(* CoDeSys 2.3.9.47 project: gym.prx *)
(* Libraries: TcBaseBX.lbx 10.5.06 08:50:20, TcSystemBX.lbx 11.6.12 13:56:16, standard.lbx 5.12.03 08:02:30, TcEIB.lbx 16.5.14 14:12:22, TcBABasicBX.lbx 22.7.15 15:46:56 *)

(* Task configuration *)
TASK Standard (PRIORITY := 0, INTERVAL := T#20ms);
	MAIN
END_TASK

(* Global variable list: KNX *)
VAR_GLOBAL
	fb_KL6301_0:								KL6301;


	fb_gym01_send_status_ex: 					EIB_BIT_SEND_EX;
	fb_gym02_send_status_ex: 					EIB_BIT_SEND_EX;
	fb_training01_send_status_ex: 				EIB_BIT_SEND_EX;
	fb_training02_send_status_ex: 				EIB_BIT_SEND_EX;
	fb_training03_send_status_ex: 				EIB_BIT_SEND_EX;
	fb_gym_stairs_bra_send_status_ex: 			EIB_BIT_SEND_EX;
	fb_pool_hall_spotlight_send_status_ex: 		EIB_BIT_SEND_EX;
	fb_pool_hall_LED_send_status_ex: 			EIB_BIT_SEND_EX;

	fb_pool_light_send_status_ex: 				EIB_BIT_SEND_EX;
	fb_sphere_ceiling_light_send_status_ex: 		EIB_BIT_SEND_EX;
	fb_sphere_light_send_status_ex: 			EIB_BIT_SEND_EX;
	fb_gym_cinema_bra_send_status_ex: 		EIB_BIT_SEND_EX;
	fb_gym_shower01_light_send_status_ex: 		EIB_BIT_SEND_EX;
	fb_gym_shower02_light_send_status_ex: 		EIB_BIT_SEND_EX;
	fb_gym_WC_corridor_send_status_ex: 		EIB_BIT_SEND_EX;
	fb_gym_stairs_light_send_status_ex: 			EIB_BIT_SEND_EX;

	fb_gym_WC_light_send_status_ex: 			EIB_BIT_SEND_EX;
	fb_training_light_send_status_ex: 			EIB_BIT_SEND_EX;
	fb_gym_light_send_status_ex: 				EIB_BIT_SEND_EX;

	fb_gym_all_send_status_ex: 				EIB_BIT_SEND_EX;
	fb_training_all_send_status_ex: 				EIB_BIT_SEND_EX;
	fb_training_1column_send_status_ex: 		EIB_BIT_SEND_EX;
	fb_pool_inwater_send_status_ex: 			EIB_BIT_SEND_EX;


	fb_outside_bigBulbs_send_status_ex:		EIB_BIT_SEND_EX;
	fb_outside_smallBulbs_send_status_ex:		EIB_BIT_SEND_EX;
	fb_outside_pingPongTable_send_status_ex:	EIB_BIT_SEND_EX;
	fb_outside_plantsLightning_send_status_ex:	EIB_BIT_SEND_EX;

	fb_pool_floor_heating_pump_send_status_ex:	EIB_BIT_SEND_EX;
	fb_gym_floor_heating_pump_send_status_ex:	EIB_BIT_SEND_EX;
	fb_vent_heating_pump_send_status_ex:		EIB_BIT_SEND_EX;
	fb_heating_pump_send_status_ex:			EIB_BIT_SEND_EX;


	fb_pool_floor_heating_pump_read:			EIB_BIT_REC ;
	fb_gym_floor_heating_pump_read:			EIB_BIT_REC ;
	fb_vent_heating_pump_read:				EIB_BIT_REC ;
	fb_heating_pump_read:					EIB_BIT_REC ;

	fb_gym01_read: 					EIB_BIT_REC;
	fb_gym02_read: 					EIB_BIT_REC;
	fb_training01_read:				EIB_BIT_REC;
	fb_training02_read:				EIB_BIT_REC;
	fb_training03_read:				EIB_BIT_REC;
	fb_gym_stairs_bra_read:			EIB_BIT_REC;
	fb_pool_hall_spotlight_read:		EIB_BIT_REC;
	fb_pool_hall_LED_read:			EIB_BIT_REC;

	fb_pool_light_read:				EIB_BIT_REC;
	fb_sphere_ceiling_light_read:		EIB_BIT_REC;
	fb_sphere_light_read:				EIB_BIT_REC;
	fb_gym_cinema_bra_read:			EIB_BIT_REC;
	fb_gym_shower01_light_read:		EIB_BIT_REC;
	fb_gym_shower02_light_read:		EIB_BIT_REC;
	fb_gym_WC_corridor_read:			EIB_BIT_REC;
	fb_gym_stairs_light_read:			EIB_BIT_REC;

	fb_gym_WC_light_read:			EIB_BIT_REC;
	fb_training_light_read:				EIB_BIT_REC;
	fb_gym_light_read:				EIB_BIT_REC;
	fb_outside_bigBulbs_read:			EIB_BIT_REC;
	fb_outside_smallBulbs_read:		EIB_BIT_REC;
	fb_outside_pingPongTable_read:	EIB_BIT_REC;
	fb_outside_plantsLightning_read:	EIB_BIT_REC;

	fb_gym_all_read: 					EIB_BIT_REC;
	fb_training_all_read: 				EIB_BIT_REC;
	fb_training_1column_read: 			EIB_BIT_REC;
	fb_pool_inwater_read: 				EIB_BIT_REC;

	gym_lights					:	BOOL;


(*2/0/x*)
	pool_floor_heating_pump_adr:								EIB_GROUP_ADDR :=(MAIN:=2, SUB_MAIN:=0, NUMBER:=1);
	gym_floor_heating_pump_adr:								EIB_GROUP_ADDR :=(MAIN:=2, SUB_MAIN:=0, NUMBER:=2);
	vent_heating_pump_adr:									EIB_GROUP_ADDR :=(MAIN:=2, SUB_MAIN:=0, NUMBER:=3);
	heating_pump_adr:										EIB_GROUP_ADDR :=(MAIN:=2, SUB_MAIN:=0, NUMBER:=4);

	pool_floor_heating_pump_status_adr:						EIB_GROUP_ADDR :=(MAIN:=2, SUB_MAIN:=0, NUMBER:=101);
	gym_floor_heating_pump_status_adr:							EIB_GROUP_ADDR :=(MAIN:=2, SUB_MAIN:=0, NUMBER:=102);
	vent_heating_pump_status_adr:								EIB_GROUP_ADDR :=(MAIN:=2, SUB_MAIN:=0, NUMBER:=103);
	heating_pump_staus_adr:									EIB_GROUP_ADDR :=(MAIN:=2, SUB_MAIN:=0, NUMBER:=104);


(*2/1/x*)
	gym01_adr:												EIB_GROUP_ADDR :=(MAIN:=2, SUB_MAIN:=1, NUMBER:=1);
	gym02_adr:												EIB_GROUP_ADDR :=(MAIN:=2, SUB_MAIN:=1, NUMBER:=2);
	training01_adr:											EIB_GROUP_ADDR :=(MAIN:=2, SUB_MAIN:=1, NUMBER:=3);
	training02_adr:											EIB_GROUP_ADDR :=(MAIN:=2, SUB_MAIN:=1, NUMBER:=4);
	training03_adr:											EIB_GROUP_ADDR :=(MAIN:=2, SUB_MAIN:=1, NUMBER:=5);
	gym_stairs_bra_adr:										EIB_GROUP_ADDR :=(MAIN:=2, SUB_MAIN:=1, NUMBER:=6);
	pool_hall_spotlight_adr:									EIB_GROUP_ADDR :=(MAIN:=2, SUB_MAIN:=1, NUMBER:=7);
	pool_hall_LED_adr:										EIB_GROUP_ADDR :=(MAIN:=2, SUB_MAIN:=1, NUMBER:=8);
	pool_light_adr:											EIB_GROUP_ADDR :=(MAIN:=2, SUB_MAIN:=1, NUMBER:=9);
	sphere_ceiling_light_adr:									EIB_GROUP_ADDR :=(MAIN:=2, SUB_MAIN:=1, NUMBER:=10);
	sphere_light_adr:											EIB_GROUP_ADDR :=(MAIN:=2, SUB_MAIN:=1, NUMBER:=11);
	gym_cinema_bra_adr:										EIB_GROUP_ADDR :=(MAIN:=2, SUB_MAIN:=1, NUMBER:=12);
	gym_shower01_light_adr:									EIB_GROUP_ADDR :=(MAIN:=2, SUB_MAIN:=1, NUMBER:=13);
	gym_shower02_light_adr:									EIB_GROUP_ADDR :=(MAIN:=2, SUB_MAIN:=1, NUMBER:=14);
	gym_WC_corridor_adr:										EIB_GROUP_ADDR :=(MAIN:=2, SUB_MAIN:=1, NUMBER:=15);
	gym_stairs_light_adr:										EIB_GROUP_ADDR:= (MAIN:=2, SUB_MAIN:=1, NUMBER:=16);
	gym_WC_light_adr:										EIB_GROUP_ADDR:= (MAIN:=2, SUB_MAIN:=1, NUMBER:=17);
	training_light_adr:											EIB_GROUP_ADDR:= (MAIN:=2, SUB_MAIN:=1, NUMBER:=18);
	gym_light_adr:											EIB_GROUP_ADDR:= (MAIN:=2, SUB_MAIN:=1, NUMBER:=19);
	training_1column_light_adr: 									EIB_GROUP_ADDR:= (MAIN:=2, SUB_MAIN:=1, NUMBER:=20);
	pool_inwater_adr: 											EIB_GROUP_ADDR:= (MAIN:=2, SUB_MAIN:=1, NUMBER:=21);




	outside_bigBulbs_adr	:									EIB_GROUP_ADDR:= (MAIN:=2, SUB_MAIN:=1, NUMBER:=25);
	outside_smallBulbs_adr:									EIB_GROUP_ADDR:= (MAIN:=2, SUB_MAIN:=1, NUMBER:=26);
	outside_pingpongTable_adr:								EIB_GROUP_ADDR:= (MAIN:=2, SUB_MAIN:=1, NUMBER:=27);
	outside_plantsLightning_adr:								EIB_GROUP_ADDR:= (MAIN:=2, SUB_MAIN:=1, NUMBER:=28);


	gym01_status_adr:										EIB_GROUP_ADDR :=(MAIN:=2, SUB_MAIN:=1, NUMBER:=101);
	gym02_status_adr:										EIB_GROUP_ADDR :=(MAIN:=2, SUB_MAIN:=1, NUMBER:=102);
	training01_status_adr:										EIB_GROUP_ADDR :=(MAIN:=2, SUB_MAIN:=1, NUMBER:=103);
	training02_status_adr:										EIB_GROUP_ADDR :=(MAIN:=2, SUB_MAIN:=1, NUMBER:=104);
	training03_status_adr:										EIB_GROUP_ADDR :=(MAIN:=2, SUB_MAIN:=1, NUMBER:=105);
	gym_stairs_bra_status_adr:									EIB_GROUP_ADDR :=(MAIN:=2, SUB_MAIN:=1, NUMBER:=106);
	pool_hall_spotlight_status_adr:								EIB_GROUP_ADDR :=(MAIN:=2, SUB_MAIN:=1, NUMBER:=107);
	pool_hall_LED_status_adr:									EIB_GROUP_ADDR :=(MAIN:=2, SUB_MAIN:=1, NUMBER:=108);
	pool_light_status_adr:										EIB_GROUP_ADDR :=(MAIN:=2, SUB_MAIN:=1, NUMBER:=109);
	sphere_ceiling_light_status_adr:								EIB_GROUP_ADDR :=(MAIN:=2, SUB_MAIN:=1, NUMBER:=110);
	sphere_light_status_adr:									EIB_GROUP_ADDR :=(MAIN:=2, SUB_MAIN:=1, NUMBER:=111);
	gym_cinema_bra_status_adr:								EIB_GROUP_ADDR :=(MAIN:=2, SUB_MAIN:=1, NUMBER:=112);
	gym_shower01_light_status_adr:								EIB_GROUP_ADDR :=(MAIN:=2, SUB_MAIN:=1, NUMBER:=113);
	gym_shower02_light_status_adr:								EIB_GROUP_ADDR :=(MAIN:=2, SUB_MAIN:=1, NUMBER:=114);
	gym_WC_corridor_status_adr:								EIB_GROUP_ADDR :=(MAIN:=2, SUB_MAIN:=1, NUMBER:=115);
	gym_stairs_light_status_adr:								EIB_GROUP_ADDR:= (MAIN:=2, SUB_MAIN:=1, NUMBER:=116);
	gym_WC_light_status_adr:									EIB_GROUP_ADDR:= (MAIN:=2, SUB_MAIN:=1, NUMBER:=117);
	training_light_status_adr:									EIB_GROUP_ADDR:= (MAIN:=2, SUB_MAIN:=1, NUMBER:=118);
	gym_light_status_adr:										EIB_GROUP_ADDR:= (MAIN:=2, SUB_MAIN:=1, NUMBER:=119);
	training_1column_light_status_adr: 							EIB_GROUP_ADDR:= (MAIN:=2, SUB_MAIN:=1, NUMBER:=120);
	pool_inwater_status_adr: 									EIB_GROUP_ADDR:= (MAIN:=2, SUB_MAIN:=1, NUMBER:=121);



	outside_bigBulbs_status_adr	:							EIB_GROUP_ADDR:= (MAIN:=2, SUB_MAIN:=1, NUMBER:=125);
	outside_smallBulbs_status_adr:								EIB_GROUP_ADDR:= (MAIN:=2, SUB_MAIN:=1, NUMBER:=126);
	outside_pingPongTable_status_adr:							EIB_GROUP_ADDR:= (MAIN:=2, SUB_MAIN:=1, NUMBER:=127);
	outside_plantsLightning_status_adr:							EIB_GROUP_ADDR:= (MAIN:=2, SUB_MAIN:=1, NUMBER:=128);

END_VAR

(* Global variable list: main *)
VAR_GLOBAL
	dataDerevo: ARRAY[0..3] OF BYTE;
	dataDerevo_prev :ARRAY[0..3] OF BYTE;

	datafloor1: ARRAY[0..3] OF BYTE;
	datafloor1_prev :ARRAY[0..3] OF BYTE;



	ads_adr_derevo: STRING:='10.0.5.64.1.1';
	ads_adr_3floor: STRING:='10.0.5.63.1.1';
	ads_adr_1floor: STRING:='10.0.5.61.1.1';

	write_ads: ADSWRITE;

	bDarkOutside						AT%MX0.0:BOOL;


	iHour							AT%MB1:	BYTE;
	iMinute							AT%MB3:	BYTE;

	t_out							AT%MB6 :	 REAL;
	heartBeatTime : TIME		:= t#30m;

	eib_gym01:							 BOOL;
	eib_gym02:							 BOOL;
	eib_training01:						 BOOL;
	eib_training02:						 BOOL;
	eib_training03	:						 BOOL;
	eib_gym_stairs_bra:					 BOOL;
	eib_pool_hall_spotlight:				 BOOL;
	eib_pool_hall_LED:					 BOOL;

	eib_pool_light:						 BOOL;
	eib_sphere_ceiling_light:				 BOOL;
	eib_sphere_light:						 BOOL;
	eib_gym_cinema_bra:					 BOOL;
	eib_gym_shower01_light:				 BOOL;
	eib_gym_shower02_light:				 BOOL;
	eib_gym_WC_corridor:					 BOOL;
	eib_gym_stairs_light:					 BOOL;

	eib_gym_WC_light:					 BOOL;
	eib_training:							 BOOL;
	eib_gym:								 BOOL;

	eib_training_1column_light	:			BOOL;
	eib_pool_inwater	:					BOOL;

	eib_pool_floor_heating_pump:			BOOL ;
	eib_gym_floor_heating_pump:			BOOL ;
	eib_vent_heating_pump:				BOOL ;
	eib_heating_pump:					BOOL ;



	eib_outside_bigBulbs:					 BOOL;
	eib_outside_pingPongTable:			 BOOL;
	eib_outside_plantsLightning:			 BOOL;
	eib_outside_smallBulbs:				 BOOL;


	floor1_tambur3_light				AT %MX100.0 :BOOL;
	sw_floor1_tambur3_short			AT %MX100.1 :BOOL;
	sw_floor1_tambur3_long			AT %MX100.2 :BOOL;
	m_heating_pump					AT %MX100.3 :BOOL;

END_VAR

(* Global variable list: TwinCAT_Import *)
VAR_GLOBAL (* DO NOT CHANGE THIS SHEET MANUALLY! *)

	gym01_light				AT %QX0.0:	BOOL; (*K01*)
	training03_light			AT %QX0.1:	BOOL; (*K05*)
	gym02_light				AT %QX0.2:	BOOL; (*K02*)
	gym_stairs_bra_right		AT %QX0.3:	BOOL; (*K06*)
	training01_light			AT %QX0.4:	BOOL; (*K03*)
	gym_stairs_bra_left		AT %QX0.5:	BOOL; (*K07*)
	training02_light			AT %QX0.6:	BOOL; (*K04*)
	pool_hall_spotlight		AT %QX0.7:	BOOL; (*K08*)

	pool_hall_ceiling_LED		AT %QX1.0:	BOOL; (*K09*)
	pool_light				AT %QX1.1:	BOOL; (*K13*)
	sphere_ceiling_light		AT %QX1.2:	BOOL; (*K10*)
	gym01_2_light			AT %QX1.3:	BOOL; (*K14*)
	sphere_light01			AT %QX1.4:	BOOL; (*K11*)
	gym02_2_light			AT %QX1.5:	BOOL; (*K15*)
	gym_cinema_bra			AT %QX1.6:	BOOL; (*K12*)
	training01_2_light			AT %QX1.7:	BOOL; (*K16*)

	training02_2_light			AT %QX2.0:	BOOL; (*K17*)
	gym_shower02_light		AT %QX2.1:	BOOL; (*K21*)
	training03_2_light			AT %QX2.2:	BOOL; (*K18*)
	gym_WC_light			AT %QX2.3:	BOOL; (*K22*)
	gym_shower01_light		AT %QX2.4:	BOOL; (*K19*)
	gym_stairs_light			AT %QX2.5:	BOOL; (*K23*)
	gym_WC_corridor			AT %QX2.6:	BOOL; (*K20*)
	sphere_light02			AT %QX2.7:	BOOL; (*K24*)

	pool_hall_LED			AT %QX3.0:	BOOL; (*K25*)
	outside_smallBulbs		AT %QX3.1:	BOOL;
	gym_cinema_TEMPORARY_light	AT %QX3.2:	BOOL; (*K26*)
	outside_bigBulbs			AT %QX3.3:	BOOL;
	Term_5_KL2408_5_Output	AT %QX3.4:	BOOL;
	outside_plantsLightning	AT %QX3.5:	BOOL;
	Term_5_KL2408_7_Output	AT %QX3.6:	BOOL;
	outside_pingPongTable	AT %QX3.7:	BOOL;

	out_5_1					AT %QX4.0:	BOOL; (**)
	fancoil_low_speed		AT %QX4.1:	BOOL; (*engineering K01*)
	out_5_3					AT %QX4.2:	BOOL; (**)
	fancoil_med_speed		AT %QX4.3:	BOOL; (*engineering K02*)
	out_5_5					AT %QX4.4:	BOOL; (**)
	fancoil_high_speed		AT %QX4.5:	BOOL; (*engineering K03*)
	out_5_7					AT %QX4.6:	BOOL; (**)
	pool_floor_heating_pump	AT %QX4.7:	BOOL; (*engineering K04*)

	heating_pump			AT %QX5.0:	BOOL; (*engineering K05*)
	storage_light				AT %QX5.1:	BOOL; (*engineering K09*)
	gym_floor_heating_pump	AT %QX5.2:	BOOL; (*engineering K06*)
	heating_room_light		AT %QX5.3:	BOOL; (*engineering K10*)
	vent_heating_pump		AT %QX5.4:	BOOL; (*engineering K07*)
	heating_storage_fan		AT %QX5.5:	BOOL; (*engineering K11*)
	out_6_7					AT %QX5.6:	BOOL; (*engineering K08*)
	pool_inwater				AT %QX5.7:	BOOL; (*engineering K12*)

	out_7_1					AT %QX6.0:	BOOL; (**)
	out_7_2					AT %QX6.1:	BOOL; (**)
	out_7_3					AT %QX6.2:	BOOL; (**)
	out_7_4					AT %QX6.3:	BOOL; (**)
	out_7_5					AT %QX6.4:	BOOL; (**)
	out_7_6					AT %QX6.5:	BOOL; (**)
	out_7_7					AT %QX6.6:	BOOL; (**)
	out_7_8					AT %QX6.7:	BOOL; (**)

	sw_02_1					AT %IX0.0:	BOOL;
	sw_01_1_2				AT %IX0.1:	BOOL;
	sw_02_2					AT %IX0.2:	BOOL;
	Term_6_KL1408_4_Input	AT %IX0.3:	BOOL;
	sw_03_1					AT %IX0.4:	BOOL;
	sw_01_1_1				AT %IX0.5:	BOOL;
	sw_01_2_1				AT %IX0.6:	BOOL;
	sw_07_1_2				AT %IX0.7:	BOOL;

	sw_07_2_2				AT %IX1.0:	BOOL;
	sw_14_1_1				AT %IX1.1:	BOOL;
	sw_07_2_1				AT %IX1.2:	BOOL;
	sw_14_1_2				AT %IX1.3:	BOOL;
	sw_07_1_1				AT %IX1.4:	BOOL;
	sw_14_2_2				AT %IX1.5:	BOOL;
	Term_7_KL1408_7_Input	AT %IX1.6:	BOOL;
	sw_14_2_1				AT %IX1.7:	BOOL;

	sw_14_3_1				AT %IX2.0:	BOOL;
	sw_09_2_2				AT %IX2.1:	BOOL;
	sw_14_3_2				AT %IX2.2:	BOOL;
	sw_09_3_1				AT %IX2.3:	BOOL;
	sw_09_1_1				AT %IX2.4:	BOOL;
	sw_09_3_2				AT %IX2.5:	BOOL;
	sw_09_2_1				AT %IX2.6:	BOOL;
	sw_09_1_2				AT %IX2.7:	BOOL;

	sw_04_1					AT %IX3.0:	BOOL;
	sw_10_1					AT %IX3.1:	BOOL;
	sw_04_2					AT %IX3.2:	BOOL;
	sw_10_2					AT %IX3.3:	BOOL;
	sw_06_1					AT %IX3.4:	BOOL;
	sw_05_2					AT %IX3.5:	BOOL;
	sw_06_2					AT %IX3.6:	BOOL;
	sw_05_1					AT %IX3.7:	BOOL;

	sw_12_1					AT %IX4.0:	BOOL;
	Term_10_KL1408_2_Input	AT %IX4.1:	BOOL;
	sw_12_2					AT %IX4.2:	BOOL;
	Term_10_KL1408_4_Input	AT %IX4.3:	BOOL;
	Term_10_KL1408_5_Input	AT %IX4.4:	BOOL;
	Term_10_KL1408_6_Input	AT %IX4.5:	BOOL;
	Term_10_KL1408_7_Input	AT %IX4.6:	BOOL;
	Term_10_KL1408_8_Input	AT %IX4.7:	BOOL;

	KL6301_IN_0 				AT %IB100: ARRAY[1..24] OF BYTE;
	KL6301_OUT_0 			AT %QB100: ARRAY[1..24] OF BYTE;

END_VAR

(* POU MAIN, ST *)
PROGRAM MAIN
VAR
	i,j:INT;
	write:BOOL;
	heartBeat: TP;
	i1: INT;
	j1: INT;
	write1: BOOL;
	sw_02_1_short_pulse:TP;
	sw_02_1_long_pulse:TP;
	sw_02_2_short_pulse:TP;
	sw_02_2_long_pulse:TP;
	sw_01_2_short_pulse:TP;
	sw_01_2_long_pulse:TP;

	sw_03_1_short_pulse: TP;
	sw_03_1_long_pulse: TP;
	init: BOOL := TRUE;
END_VAR
heartBeat(IN:= NOT heartBeat.Q, PT:=t#5s);

EIB;
ADS_Communication;
(*Light.knx_triggers;*)
Light;
Light.outsideLight;
engineering;
(*Counters;*)
write_ADSdata;
END_PROGRAM
ACTION write_ADSdata:
	sw_02_1_short_pulse(IN:= Light.fb_sw_02_1.bShortClick, pt:=t#500ms);
	sw_02_1_long_pulse(IN:= Light.fb_sw_02_1.bLongClick, pt:=t#500ms);
	sw_02_2_short_pulse(IN:= Light.fb_sw_02_2.bShortClick, pt:=t#500ms);
	sw_02_2_long_pulse(IN:= Light.fb_sw_02_2.bLongClick, pt:=t#500ms);
	sw_01_2_short_pulse(IN:= Light.fb_sw_01_2_1.bShortClick, pt:=t#500ms);
	sw_01_2_long_pulse(IN:= Light.fb_sw_01_2_1.bLongClick, pt:=t#500ms);

	sw_03_1_short_pulse(IN:= Light.fb_sw_03_1.bShortClick, pt:=t#500ms);
	sw_03_1_long_pulse(IN:= Light.fb_sw_03_1.bLongClick, pt:=t#500ms);


	datafloor1[0].0 := sw_02_1_short_pulse.Q;
	datafloor1[0].1 := sw_02_1_long_pulse.Q;
	datafloor1[0].2 := sw_02_2_short_pulse.Q;
	datafloor1[0].3 := sw_02_2_long_pulse.Q;
	datafloor1[0].4 := gym_stairs_bra_left;
	datafloor1[0].5 := sw_01_2_short_pulse.Q;
	datafloor1[0].6 := sw_01_2_long_pulse.Q;
	datafloor1[0].7 := sw_03_1_short_pulse.Q;
	datafloor1[1].0 := sw_03_1_long_pulse.Q;

FOR i:=0 TO (SIZEOF(dataDerevo))-1 DO
	IF dataDerevo[i]<>dataDerevo_prev[i]  THEN
		write:=TRUE;
		EXIT;
	ELSE
		write:=FALSE;
	END_IF
END_FOR


FOR j:=0 TO (SIZEOF(dataDerevo))-1 DO
	dataDerevo_prev[j]:=dataDerevo[j];
END_FOR

FOR i1:=0 TO (SIZEOF(dataFloor1))-1 DO
	IF dataFloor1[i1]<>dataFloor1_prev[i1]  THEN
		write1:=TRUE;
		EXIT;
	ELSE
		write1:=FALSE;
	END_IF
END_FOR


FOR j1:=0 TO (SIZEOF(dataFloor1))-1 DO
	dataFloor1_prev[j1]:=dataFloor1[j1];
END_FOR
END_ACTION

(* POU EIB, ST *)
PROGRAM EIB
VAR

	eib_send_mode_gym:INT;
	eib_send_cyclical_start_gym: BOOL;

	floors:INT;
	i:INT;
	fb_sending_floor_order:CTU;
	fb_heartbeat_timer:TON;
	fb_sending_time_frame:TOF;

	fb_start_delay:TP;

END_VAR
fb_start_delay(IN:=  SYSTEMTASKINFOARR[1].firstCycle, PT:=t#10s);

(*EIB*)
fb_heartbeat_timer(in:=NOT  fb_heartbeat_timer.Q, pt:=heartBeatTime);
fb_sending_time_frame(in:=fb_heartbeat_timer.Q, pt:=t#50ms);
fb_sending_floor_order(cu:=fb_heartbeat_timer.Q, pv:=4,reset:=fb_sending_floor_order.CV >4, CV=>floors);

IF NOT fb_start_delay.Q THEN
	eib_send_mode_gym:=2;
ELSE
	eib_send_mode_gym:=0;
	eib_send_cyclical_start_gym:=TRUE;
END_IF


CASE floors OF
1:
	eib_send_mode_gym:=2*BOOL_TO_INT(NOT (fb_sending_time_frame.Q)); (*0-manual*)
	IF fb_heartbeat_timer.Q THEN
		eib_send_cyclical_start_gym:=FALSE;
	ELSE
		eib_send_cyclical_start_gym:=TRUE;
	END_IF

	heartBeatTime := t#10m;
END_CASE


fb_KL6301_0.iMode:=1;
CASE i OF
0:	(* EIB Address 1.1.2 *)
	fb_KL6301_0.EIB_PHYS_ADDR.Area:=1;
	fb_KL6301_0.EIB_PHYS_ADDR.Line:=1;
	fb_KL6301_0.EIB_PHYS_ADDR.Device:=2;
	(* Filter 1 *)
	fb_KL6301_0.EIB_GROUP_FILTER[1].GROUP_ADDR.MAIN:=2;
	fb_KL6301_0.EIB_GROUP_FILTER[1].GROUP_ADDR.SUB_MAIN:=0;
	fb_KL6301_0.EIB_GROUP_FILTER[1].GROUP_ADDR.NUMBER:=0;
	fb_KL6301_0.EIB_GROUP_FILTER[1].GROUP_LEN:=31;
	(* Filter 2*)
	fb_KL6301_0.EIB_GROUP_FILTER[2].GROUP_ADDR.MAIN:=2;
	fb_KL6301_0.EIB_GROUP_FILTER[2].GROUP_ADDR.SUB_MAIN:=1;
	fb_KL6301_0.EIB_GROUP_FILTER[2].GROUP_ADDR.NUMBER:=0;
	fb_KL6301_0.EIB_GROUP_FILTER[2].GROUP_LEN:=31;
	(* Filter 3*)
	fb_KL6301_0.EIB_GROUP_FILTER[3].GROUP_ADDR.MAIN:=2;
	fb_KL6301_0.EIB_GROUP_FILTER[3].GROUP_ADDR.SUB_MAIN:=2;
	fb_KL6301_0.EIB_GROUP_FILTER[3].GROUP_ADDR.NUMBER:=0;
	fb_KL6301_0.EIB_GROUP_FILTER[3].GROUP_LEN:=31;
	(* Filter 4 *)
	fb_KL6301_0.EIB_GROUP_FILTER[4].GROUP_ADDR.MAIN:=2;
	fb_KL6301_0.EIB_GROUP_FILTER[4].GROUP_ADDR.SUB_MAIN:=3;
	fb_KL6301_0.EIB_GROUP_FILTER[4].GROUP_ADDR.NUMBER:=0;
	fb_KL6301_0.EIB_GROUP_FILTER[4].GROUP_LEN:=31;
	(* Filter 5*)
	fb_KL6301_0.EIB_GROUP_FILTER[5].GROUP_ADDR.MAIN:=2;
	fb_KL6301_0.EIB_GROUP_FILTER[5].GROUP_ADDR.SUB_MAIN:=4;
	fb_KL6301_0.EIB_GROUP_FILTER[5].GROUP_ADDR.NUMBER:=0;
	fb_KL6301_0.EIB_GROUP_FILTER[5].GROUP_LEN:=31;
	(* Filter 6*)
	fb_KL6301_0.EIB_GROUP_FILTER[6].GROUP_ADDR.MAIN:=2;
	fb_KL6301_0.EIB_GROUP_FILTER[6].GROUP_ADDR.SUB_MAIN:=5;
	fb_KL6301_0.EIB_GROUP_FILTER[6].GROUP_ADDR.NUMBER:=0;
	fb_KL6301_0.EIB_GROUP_FILTER[6].GROUP_LEN:=31;
	(* Filter 7*)
	fb_KL6301_0.EIB_GROUP_FILTER[7].GROUP_ADDR.MAIN:=2;
	fb_KL6301_0.EIB_GROUP_FILTER[7].GROUP_ADDR.SUB_MAIN:=6;
	fb_KL6301_0.EIB_GROUP_FILTER[7].GROUP_ADDR.NUMBER:=0;
	fb_KL6301_0.EIB_GROUP_FILTER[7].GROUP_LEN:=31;
	(* Filter 8*)
	fb_KL6301_0.EIB_GROUP_FILTER[8].GROUP_ADDR.MAIN:=1;
	fb_KL6301_0.EIB_GROUP_FILTER[8].GROUP_ADDR.SUB_MAIN:=7;
	fb_KL6301_0.EIB_GROUP_FILTER[8].GROUP_ADDR.NUMBER:=0;
	fb_KL6301_0.EIB_GROUP_FILTER[8].GROUP_LEN:=31;

	fb_KL6301_0.bActivate :=TRUE; 	(*Start EIB Functionblock*)
	IF fb_KL6301_0.bReady THEN	(*Wait until the fb is ready *)
		IF NOT fb_KL6301_0.bError THEN
			i:=1;  (* EIB functionblock is now ready to send and receive *)
		ELSE
			i:=100; (* EIB ERROR*)
		END_IF
	END_IF
1:	;
100:	;(*ERROR EIB*)
END_CASE

fb_KL6301_0(
	idx:=1,								(* for every KL6301 an other idx number
										Example KL6301 terminal 1 - idx=1 , KL6301 termnal 2 -idx=3,... max. 64 *)
	KL6301_IN:=KL6301_IN_0,				(* Terminal variable - address IN *)
	KL6301_OUT:=KL6301_OUT_0 );			(* Terminal variable - address OUT *)



gym_and_outside;
END_PROGRAM
ACTION gym_and_outside:
fb_gym01_read(
	strData_Rec:=fb_KL6301_0.str_Data_Rec,
	Group_Address:=gym01_adr,
	);
IF NOT fb_gym01_read.bDataReceive THEN
	eib_gym01 := fb_gym01_read.bData;
END_IF

fb_gym02_read(
	strData_Rec:=fb_KL6301_0.str_Data_Rec,
	Group_Address:=gym02_adr,
	);
IF NOT fb_gym02_read.bDataReceive THEN
	eib_gym02 := fb_gym02_read.bData;
END_IF

fb_gym_all_read(
	strData_Rec:=fb_KL6301_0.str_Data_Rec,
	Group_Address:=gym_light_adr,
	);
IF NOT fb_gym_all_read.bDataReceive THEN
	eib_gym := fb_gym_all_read.bData;
	eib_gym01 := fb_gym_all_read.bData;
	eib_gym02 := fb_gym_all_read.bData;
END_IF

fb_training01_read(
	strData_Rec:=fb_KL6301_0.str_Data_Rec,
	Group_Address:=training01_adr,
	);
IF NOT fb_training01_read.bDataReceive THEN
	eib_training01 := fb_training01_read.bData;
END_IF

fb_training02_read(
	strData_Rec:=fb_KL6301_0.str_Data_Rec,
	Group_Address:=training02_adr,
	);
IF NOT fb_training02_read.bDataReceive THEN
	eib_training02 := fb_training02_read.bData;
END_IF

fb_training03_read(
	strData_Rec:=fb_KL6301_0.str_Data_Rec,
	Group_Address:=training03_adr
	);
IF NOT fb_training03_read.bDataReceive THEN
	eib_training03 := fb_training03_read.bData;
END_IF

fb_training_all_read(
	strData_Rec:=fb_KL6301_0.str_Data_Rec,
	Group_Address:=training_light_adr
	);
IF NOT fb_training_all_read.bDataReceive THEN
	eib_training01 := fb_training_all_read.bData;
	eib_training02 := fb_training_all_read.bData;
	eib_training03 := fb_training_all_read.bData;
	eib_training_1column_light:= fb_training_all_read.bData;
	eib_training := fb_training_all_read.bData;
END_IF


fb_training_1column_read(
	strData_Rec:=fb_KL6301_0.str_Data_Rec,
	Group_Address:=training_1column_light_adr,
	);
IF NOT fb_training_1column_read.bDataReceive THEN
	eib_training_1column_light := fb_training_1column_read.bData;
END_IF

fb_gym_stairs_bra_read(
	strData_Rec:=fb_KL6301_0.str_Data_Rec,
	Group_Address:=gym_stairs_bra_adr,
	bData=>eib_gym_stairs_bra
	);

fb_pool_hall_spotlight_read(
	strData_Rec:=fb_KL6301_0.str_Data_Rec,
	Group_Address:=pool_hall_spotlight_adr,
	bData=>eib_pool_hall_spotlight,
	);

fb_pool_hall_LED_read(
	strData_Rec:=fb_KL6301_0.str_Data_Rec,
	Group_Address:=pool_hall_LED_adr,
	bData=>eib_pool_hall_LED
	);

fb_pool_light_read(
	strData_Rec:=fb_KL6301_0.str_Data_Rec,
	Group_Address:=pool_light_adr,
	bData=>eib_pool_light
	);

fb_pool_inwater_read(
	strData_Rec:=fb_KL6301_0.str_Data_Rec,
	Group_Address:=pool_inwater_adr,
	bData=>eib_pool_inwater
	);

fb_sphere_ceiling_light_read(
	strData_Rec:=fb_KL6301_0.str_Data_Rec,
	Group_Address:=sphere_ceiling_light_adr,
	bData=>eib_sphere_ceiling_light
	);

fb_sphere_light_read(
	strData_Rec:=fb_KL6301_0.str_Data_Rec,
	Group_Address:=sphere_light_adr,
	bData=>eib_sphere_light
	);

fb_gym_cinema_bra_read(
	strData_Rec:=fb_KL6301_0.str_Data_Rec,
	Group_Address:=gym_cinema_bra_adr,
	bData=>eib_gym_cinema_bra
	);

fb_gym_shower01_light_read(
	strData_Rec:=fb_KL6301_0.str_Data_Rec,
	Group_Address:=gym_shower01_light_adr,
	bData=>eib_gym_shower01_light
	);

fb_gym_shower02_light_read(
	strData_Rec:=fb_KL6301_0.str_Data_Rec,
	Group_Address:=gym_shower02_light_adr,
	bData=>eib_gym_shower02_light
);

fb_gym_WC_corridor_read(
	strData_Rec:=fb_KL6301_0.str_Data_Rec,
	Group_Address:=gym_WC_corridor_adr,
	bData=>eib_gym_WC_corridor
	);

fb_gym_stairs_light_read(
	strData_Rec:=fb_KL6301_0.str_Data_Rec,
	Group_Address:=gym_stairs_bra_adr,
	bData=>eib_gym_stairs_bra
	);

fb_gym_WC_light_read(
	strData_Rec:=fb_KL6301_0.str_Data_Rec,
	Group_Address:=gym_WC_light_adr,
	bData=>eib_gym_WC_light
	);


fb_pool_floor_heating_pump_read(
	strData_Rec:=fb_KL6301_0.str_Data_Rec,
	Group_Address:=pool_floor_heating_pump_adr,
	bData=>eib_pool_floor_heating_pump
	);

fb_gym_floor_heating_pump_read(
	strData_Rec:=fb_KL6301_0.str_Data_Rec,
	Group_Address:=gym_floor_heating_pump_adr,
	bData=>eib_gym_floor_heating_pump
	);

fb_vent_heating_pump_read(
	strData_Rec:=fb_KL6301_0.str_Data_Rec,
	Group_Address:=vent_heating_pump_adr,
	bData=>eib_vent_heating_pump
	);

fb_heating_pump_read(
	strData_Rec:=fb_KL6301_0.str_Data_Rec,
	Group_Address:=heating_pump_adr,
	bData=>eib_heating_pump
	);


fb_outside_bigBulbs_read(
	strData_Rec:=fb_KL6301_0.str_Data_Rec,
	Group_Address:=outside_bigBulbs_adr
);
IF NOT  fb_outside_Bigbulbs_read.bDataReceive THEN
	eib_outside_bigBulbs:= fb_outside_bigBulbs_read.bdata;
END_IF

fb_outside_pingPongTable_read(
	strData_Rec:=fb_KL6301_0.str_Data_Rec,
	Group_Address:=outside_pingPongTable_adr
);
IF NOT  fb_outside_pingPongTable_read.bDataReceive THEN
	eib_outside_pingPongTable:= fb_outside_pingPongTable_read.bdata;
END_IF

fb_outside_plantsLightning_read(
	strData_Rec:=fb_KL6301_0.str_Data_Rec,
	Group_Address:=outside_plantsLightning_adr
	);
IF NOT  fb_outside_plantsLightning_read.bDataReceive THEN
	eib_outside_plantsLightning:= fb_outside_plantsLightning_read.bdata;
END_IF

fb_outside_smallBulbs_read(
	strData_Rec:=fb_KL6301_0.str_Data_Rec,
	Group_Address:=outside_smallBulbs_adr
);
IF NOT  fb_outside_smallBulbs_read.bDataReceive THEN
	eib_outside_smallBulbs:= fb_outside_smallBulbs_read.bdata;
END_IF

(*sending*)

fb_gym01_send_status_ex(
	imode:=eib_send_mode_gym,
	bStart:=eib_send_cyclical_start_gym,
	str_Rec:=fb_KL6301_0.str_Data_Rec,
	bData:=gym01_light OR gym01_2_light,
	Group_Address:=gym01_status_adr
	);

fb_gym02_send_status_ex(
	imode:=eib_send_mode_gym,
	bStart:=eib_send_cyclical_start_gym,
	str_Rec:=fb_KL6301_0.str_Data_Rec,
	bData:=gym02_light OR gym02_2_light,
	Group_Address:=gym02_status_adr
	);
fb_gym_light_send_status_ex(
	imode:=eib_send_mode_gym,
	bStart:=eib_send_cyclical_start_gym,
	str_Rec:=fb_KL6301_0.str_Data_Rec,
	bData:=gym02_2_light OR gym01_2_light,
	Group_Address:=gym_light_status_adr
	);

fb_training01_send_status_ex(
	imode:=eib_send_mode_gym,
	bStart:=eib_send_cyclical_start_gym,
	str_Rec:=fb_KL6301_0.str_Data_Rec,
	bData:=training01_light OR training01_2_light,
	Group_Address:=training01_status_adr
	);

fb_training02_send_status_ex(
	imode:=eib_send_mode_gym,
	bStart:=eib_send_cyclical_start_gym,
	str_Rec:=fb_KL6301_0.str_Data_Rec,
	bData:=training02_light OR training02_2_light,
	Group_Address:=training02_status_adr
	);
fb_gym_stairs_bra_send_status_ex(
	imode:=eib_send_mode_gym,
	bStart:=eib_send_cyclical_start_gym,
	str_Rec:=fb_KL6301_0.str_Data_Rec,
	bData:=gym_stairs_bra_left,
	Group_Address:=gym_stairs_bra_status_adr
	);
fb_training03_send_status_ex(
	imode:=eib_send_mode_gym,
	bStart:=eib_send_cyclical_start_gym,
	str_Rec:=fb_KL6301_0.str_Data_Rec,
	bData:=training03_light OR training03_2_light,
	Group_Address:=training03_status_adr
	);
fb_training_light_send_status_ex(
	imode:=eib_send_mode_gym,
	bStart:=eib_send_cyclical_start_gym,
	str_Rec:=fb_KL6301_0.str_Data_Rec,
	bData:=training01_2_light AND training03_2_light,
	Group_Address:=training_light_status_adr
	);
fb_training_1column_send_status_ex(
	imode:=eib_send_mode_gym,
	bStart:=eib_send_cyclical_start_gym,
	str_Rec:=fb_KL6301_0.str_Data_Rec,
	bData:=training01_2_light,
	Group_Address:=training_1column_light_status_adr
	);

fb_pool_hall_spotlight_send_status_ex(
	imode:=eib_send_mode_gym,
	bStart:=eib_send_cyclical_start_gym,
	str_Rec:=fb_KL6301_0.str_Data_Rec,
	bData:=pool_hall_spotlight,
	Group_Address:=pool_hall_spotlight_status_adr
	);

fb_pool_hall_LED_send_status_ex(
	imode:=eib_send_mode_gym,
	bStart:=eib_send_cyclical_start_gym,
	str_Rec:=fb_KL6301_0.str_Data_Rec,
	bData:=pool_hall_LED,
	Group_Address:=pool_hall_LED_status_adr
	);

fb_pool_light_send_status_ex(
	imode:=eib_send_mode_gym,
	bStart:=eib_send_cyclical_start_gym,
	str_Rec:=fb_KL6301_0.str_Data_Rec,
	bData:=pool_light,
	Group_Address:=pool_light_status_adr
	);

fb_pool_inwater_send_status_ex(
	imode:=eib_send_mode_gym,
	bStart:=eib_send_cyclical_start_gym,
	str_Rec:=fb_KL6301_0.str_Data_Rec,
	bData:=pool_inwater,
	Group_Address:=pool_inwater_status_adr
	);

fb_sphere_ceiling_light_send_status_ex(
	imode:=eib_send_mode_gym,
	bStart:=eib_send_cyclical_start_gym,
	str_Rec:=fb_KL6301_0.str_Data_Rec,
	bData:=sphere_ceiling_light,
	Group_Address:=sphere_ceiling_light_status_adr
	);

fb_sphere_light_send_status_ex(
	imode:=eib_send_mode_gym,
	bStart:=eib_send_cyclical_start_gym,
	str_Rec:=fb_KL6301_0.str_Data_Rec,
	bData:=sphere_light01,
	Group_Address:=sphere_light_status_adr
	);

fb_gym_cinema_bra_send_status_ex(
	imode:=eib_send_mode_gym,
	bStart:=eib_send_cyclical_start_gym,
	str_Rec:=fb_KL6301_0.str_Data_Rec,
	bData:=gym_cinema_bra,
	Group_Address:=gym_cinema_bra_status_adr
	);

fb_gym_shower01_light_send_status_ex(
	imode:=eib_send_mode_gym,
	bStart:=eib_send_cyclical_start_gym,
	str_Rec:=fb_KL6301_0.str_Data_Rec,
	bData:=gym_shower01_light,
	Group_Address:=gym_shower01_light_status_adr
	);

fb_gym_shower02_light_send_status_ex(
	imode:=eib_send_mode_gym,
	bStart:=eib_send_cyclical_start_gym,
	str_Rec:=fb_KL6301_0.str_Data_Rec,
	bData:=gym_shower02_light,
	Group_Address:=gym_shower02_light_status_adr
	);

fb_gym_WC_corridor_send_status_ex(
	imode:=eib_send_mode_gym,
	bStart:=eib_send_cyclical_start_gym,
	str_Rec:=fb_KL6301_0.str_Data_Rec,
	bData:=gym_WC_corridor,
	Group_Address:=gym_WC_corridor_status_adr
	);

fb_gym_stairs_light_send_status_ex(
	imode:=eib_send_mode_gym,
	bStart:=eib_send_cyclical_start_gym,
	str_Rec:=fb_KL6301_0.str_Data_Rec,
	bData:=gym_stairs_light,
	Group_Address:=gym_stairs_light_status_adr
	);

fb_gym_WC_light_send_status_ex(
	imode:=eib_send_mode_gym,
	bStart:=eib_send_cyclical_start_gym,
	str_Rec:=fb_KL6301_0.str_Data_Rec,
	bData:=gym_WC_light,
	Group_Address:=gym_WC_light_status_adr
	);

fb_pool_floor_heating_pump_send_status_ex(
	imode:=eib_send_mode_gym,
	bStart:=eib_send_cyclical_start_gym,
	str_Rec:=fb_KL6301_0.str_Data_Rec,
	bData:=pool_floor_heating_pump,
	Group_Address:=pool_floor_heating_pump_status_adr
	);

fb_gym_floor_heating_pump_send_status_ex(
	imode:=eib_send_mode_gym,
	bStart:=eib_send_cyclical_start_gym,
	str_Rec:=fb_KL6301_0.str_Data_Rec,
	bData:=gym_floor_heating_pump,
	Group_Address:=gym_floor_heating_pump_status_adr
	);

fb_vent_heating_pump_send_status_ex(
	imode:=eib_send_mode_gym,
	bStart:=eib_send_cyclical_start_gym,
	str_Rec:=fb_KL6301_0.str_Data_Rec,
	bData:=vent_heating_pump,
	Group_Address:=vent_heating_pump_status_adr
	);

fb_heating_pump_send_status_ex(
	imode:=eib_send_mode_gym,
	bStart:=eib_send_cyclical_start_gym,
	str_Rec:=fb_KL6301_0.str_Data_Rec,
	bData:=heating_pump,
	Group_Address:=heating_pump_staus_adr
	);

fb_outside_bigBulbs_send_status_ex(
	imode:=eib_send_mode_gym,
	bStart:=eib_send_cyclical_start_gym,
	str_Rec:=fb_KL6301_0.str_Data_Rec,
	bData:=outside_bigBulbs,
	Group_Address:=outside_bigBulbs_status_adr
	);
fb_outside_pingPongTable_send_status_ex(
	imode:=eib_send_mode_gym,
	bStart:=eib_send_cyclical_start_gym,
	str_Rec:=fb_KL6301_0.str_Data_Rec,
	bData:=outside_pingPongTable,
	Group_Address:=outside_pingPongTable_status_adr
	);

fb_outside_plantsLightning_send_status_ex(
	imode:=eib_send_mode_gym,
	bStart:=eib_send_cyclical_start_gym,
	str_Rec:=fb_KL6301_0.str_Data_Rec,
	bData:=outside_plantsLightning,
	Group_Address:=outside_plantsLightning_status_adr
	);

fb_outside_smallBulbs_send_status_ex(
	imode:=eib_send_mode_gym,
	bStart:=eib_send_cyclical_start_gym,
	str_Rec:=fb_KL6301_0.str_Data_Rec,
	bData:=outside_smallBulbs,
	Group_Address:=outside_smallBulbs_status_adr
);
END_ACTION

(* POU ADS_Communication, CFC *)
PROGRAM ADS_Communication
VAR
	fb_DerevoADSwrite: ADSWRITE;
	fb_floor1ADSwrite: ADSWRITE;

	counter_error,counter_busy: CTU;
END_VAR
VAR (* helpers for the ST form of the networks *)
	_t21 : DWORD;
	_t23 : DWORD;
	_t42 : BOOL;
	_t50 : DWORD;
	_t52 : DWORD;
	_t56 : BOOL;
END_VAR
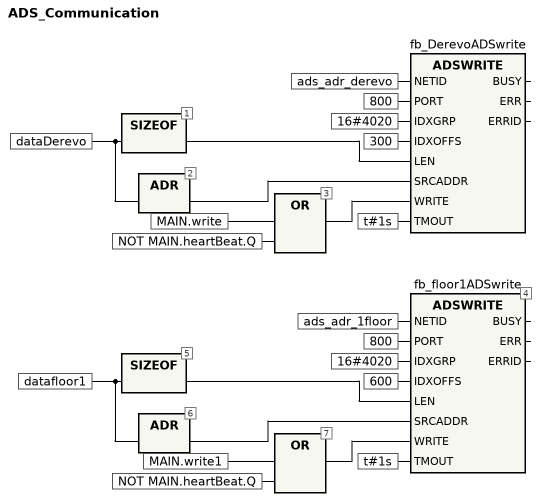
_CFC_ (* Continuous Function Chart, elements in execution order *)
#0 fb_DerevoADSwrite:ADSWRITE(NETID: ads_adr_derevo, PORT: 800, IDXGRP: 16#4020, IDXOFFS: 300, LEN: #1, SRCADDR: #2, WRITE: #3, TMOUT: t#1s)
#1 SIZEOF(dataDerevo)
#2 ADR(dataDerevo)
#3 OR(MAIN.write, NOT MAIN.heartBeat.Q)
#4 fb_floor1ADSwrite:ADSWRITE(NETID: ads_adr_1floor, PORT: 800, IDXGRP: 16#4020, IDXOFFS: 600, LEN: #5, SRCADDR: #6, WRITE: #7, TMOUT: t#1s)
#5 SIZEOF(datafloor1)
#6 ADR(datafloor1)
#7 OR(MAIN.write1, NOT MAIN.heartBeat.Q)
_END_CFC_
(* the same logic as Structured Text *)
fb_DerevoADSwrite(NETID := ads_adr_derevo, PORT := 800, IDXGRP := 16#4020, IDXOFFS := 300, LEN := _t21, SRCADDR := _t23, WRITE := _t42, TMOUT := t#1s);
_t21 := SIZEOF(dataDerevo);
_t23 := ADR(dataDerevo);
_t42 := MAIN.write OR NOT MAIN.heartBeat.Q;
fb_floor1ADSwrite(NETID := ads_adr_1floor, PORT := 800, IDXGRP := 16#4020, IDXOFFS := 600, LEN := _t50, SRCADDR := _t52, WRITE := _t56, TMOUT := t#1s);
_t50 := SIZEOF(datafloor1);
_t52 := ADR(datafloor1);
_t56 := MAIN.write1 OR NOT MAIN.heartBeat.Q;
END_PROGRAM

(* POU Light, CFC *)
PROGRAM Light
VAR
	(*switches*)

	fb_sw_01_1_2	:	FB_ShortLongClick;
	fb_sw_01_1_1	:	FB_ShortLongClick;
	fb_sw_01_2_1	:	FB_ShortLongClick;
	fb_sw_07_1_1	:	FB_ShortLongClick;
	fb_sw_07_2_1	:	FB_ShortLongClick;
	fb_sw_14_1_1	:	FB_ShortLongClick;
	fb_sw_14_1_2	:	FB_ShortLongClick;
	fb_sw_14_2_2	:	FB_ShortLongClick;
	fb_sw_14_2_1	:	FB_ShortLongClick;
	fb_sw_14_3_1	:	FB_ShortLongClick;
	fb_sw_09_2_2	:	FB_ShortLongClick;
	fb_sw_14_3_2	:	FB_ShortLongClick;
	fb_sw_09_3_1	:	FB_ShortLongClick;
	fb_sw_09_1_1	:	FB_ShortLongClick;
	fb_sw_09_3_2	:	FB_ShortLongClick;
	fb_sw_09_2_1	:	FB_ShortLongClick;
	fb_sw_09_1_2	:	FB_ShortLongClick;
	fb_sw_04_1	:	FB_ShortLongClick;
	fb_sw_04_2	:	FB_ShortLongClick;
	fb_sw_06_1	:	FB_ShortLongClick;
	fb_sw_06_2	:	FB_ShortLongClick;

	longPressTimeout	:	TIME := t#500ms;

	(*Lights*)
	fb_gym01_light			: FB_Light;
	fb_gym02_light			: FB_Light;
	fb_training01_light			: FB_Light;
	fb_training02_light			: FB_Light;
	fb_training03_light			: FB_Light;
	fb_gym_stairs_bra			: FB_Light;
	fb_pool_hall_spotlight		: FB_Light;
	fb_pool_hall_LED			: FB_Light;
	fb_pool_light				: FB_Light;
	fb_sphere_ceiling_light		: FB_Light;
	fb_sphere_light			: FB_Light;
	fb_gym_cinema_bra		: FB_Light;
	fb_gym_shower01_light		: FB_Light;
	fb_gym_shower02_light		: FB_Light;
	fb_gym_WC_corridor		: FB_Light;
	fb_gym_stairs_light		: FB_Light;
	fb_gym_WC_light			: FB_Light;
	fb_training_light			: FB_Light;
	fb_gym_light				: FB_Light;


	fb_cinema_temporary_light	:FB_Light;

	traning_falling_edge :F_TRIG;
	gym_falling_edge :F_TRIG;


	fb_sw_05_1: FB_ShortLongClick;
	fb_sw_05_2: FB_ShortLongClick;
	fb_training01_2_light: FB_Light;
	fb_gym_01_2_light: FB_Light;
	fb_gym01_2_light: FB_Light;


	rising_edge_eib_gym01 						:	 R_TRIG;
	rising_edge_eib_gym02 						:	 R_trig;
	rising_edge_eib_training01 					:	 R_trig;
	rising_edge_eib_training02						:	 R_trig;
	rising_edge_eib_training03						:	 R_trig;
	rising_edge_eib_gym_stairs_bra				:	 R_trig;
	rising_edge_eib_pool_hall_spotlight				:	 R_trig;
	rising_edge_eib_pool_hall_LED				:	 R_trig;

	rising_edge_eib_pool_light 					:	 R_trig;
	rising_edge_eib_sphere_ceiling_light 			:	 R_trig;
	rising_edge_eib_sphere_light 					:	 R_trig;
	rising_edge_eib_gym_cinema_bra 				:	 R_trig;
	rising_edge_eib_gym_shower01_light			:	 R_trig;
	rising_edge_eib_gym_shower02_light			:	 R_trig;
	rising_edge_eib_gym_WC_corridor				:	 R_trig;
	rising_edge_eib_gym_stairs_light 				:	 R_trig;

	rising_edge_eib_gym_WC_light 				:	 R_trig;
	rising_edge_eib_training	 					:	 R_trig;
	rising_edge_eib_gym		 					:	 R_TRIG;

	falling_edge_eib_gym01 						:	 F_TRIG;
	falling_edge_eib_gym02 						:	 F_TRIG;
	falling_edge_eib_training01 					:	 F_TRIG;
	falling_edge_eib_training02						:	 F_TRIG;
	falling_edge_eib_training03						:	 F_TRIG;
	falling_edge_eib_gym_stairs_bra				:	 F_TRIG;
	falling_edge_eib_pool_hall_spotlight				:	 F_TRIG;
	falling_edge_eib_pool_hall_LED				:	 F_TRIG;

	falling_edge_eib_pool_light 					:	 F_TRIG;
	falling_edge_eib_sphere_ceiling_light 			:	 F_TRIG;
	falling_edge_eib_sphere_light 					:	 F_TRIG;
	falling_edge_eib_gym_cinema_bra 				:	 F_TRIG;
	falling_edge_eib_gym_shower01_light			:	 F_TRIG;
	falling_edge_eib_gym_shower02_light			:	 F_TRIG;
	falling_edge_eib_gym_WC_corridor				:	 F_TRIG;
	falling_edge_eib_gym_stairs_light 				:	 F_TRIG;

	falling_edge_eib_gym_WC_light 				:	 F_TRIG;
	falling_edge_eib_training	 					:	 F_TRIG;
	falling_edge_eib_gym		 					:	 F_TRIG;

	(*timers*)
	fb_OutsideLightTimer	:TP;

	fb_pool_hall_all: FB_Light;
	pool_all_falling_edge: F_TRIG;
	pool_all_rising_edge: R_TRIG;
	pool_hall_all_rising_edge: R_TRIG;
	pool_hall_all_falling_edge: F_TRIG;
	traning_reserved_falling_edge: F_TRIG;
	fb_sw_07_1_2: FB_ShortLongClick;
	fb_sw_07_2_2: FB_ShortLongClick;
	fb_sw_02_1: FB_ShortLongClick;
	fb_sw_02_2: FB_ShortLongClick;
	fb_sw_03_1: FB_ShortLongClick;
	darkOutside_rising_edge:R_TRIG;

	darkness_correction_time_hour:INT := 20;

	pool_inwater_rising_edge: R_TRIG;
	pool_light_rising_edge: R_TRIG;
	fb_pool_inwater: FB_Light;
END_VAR
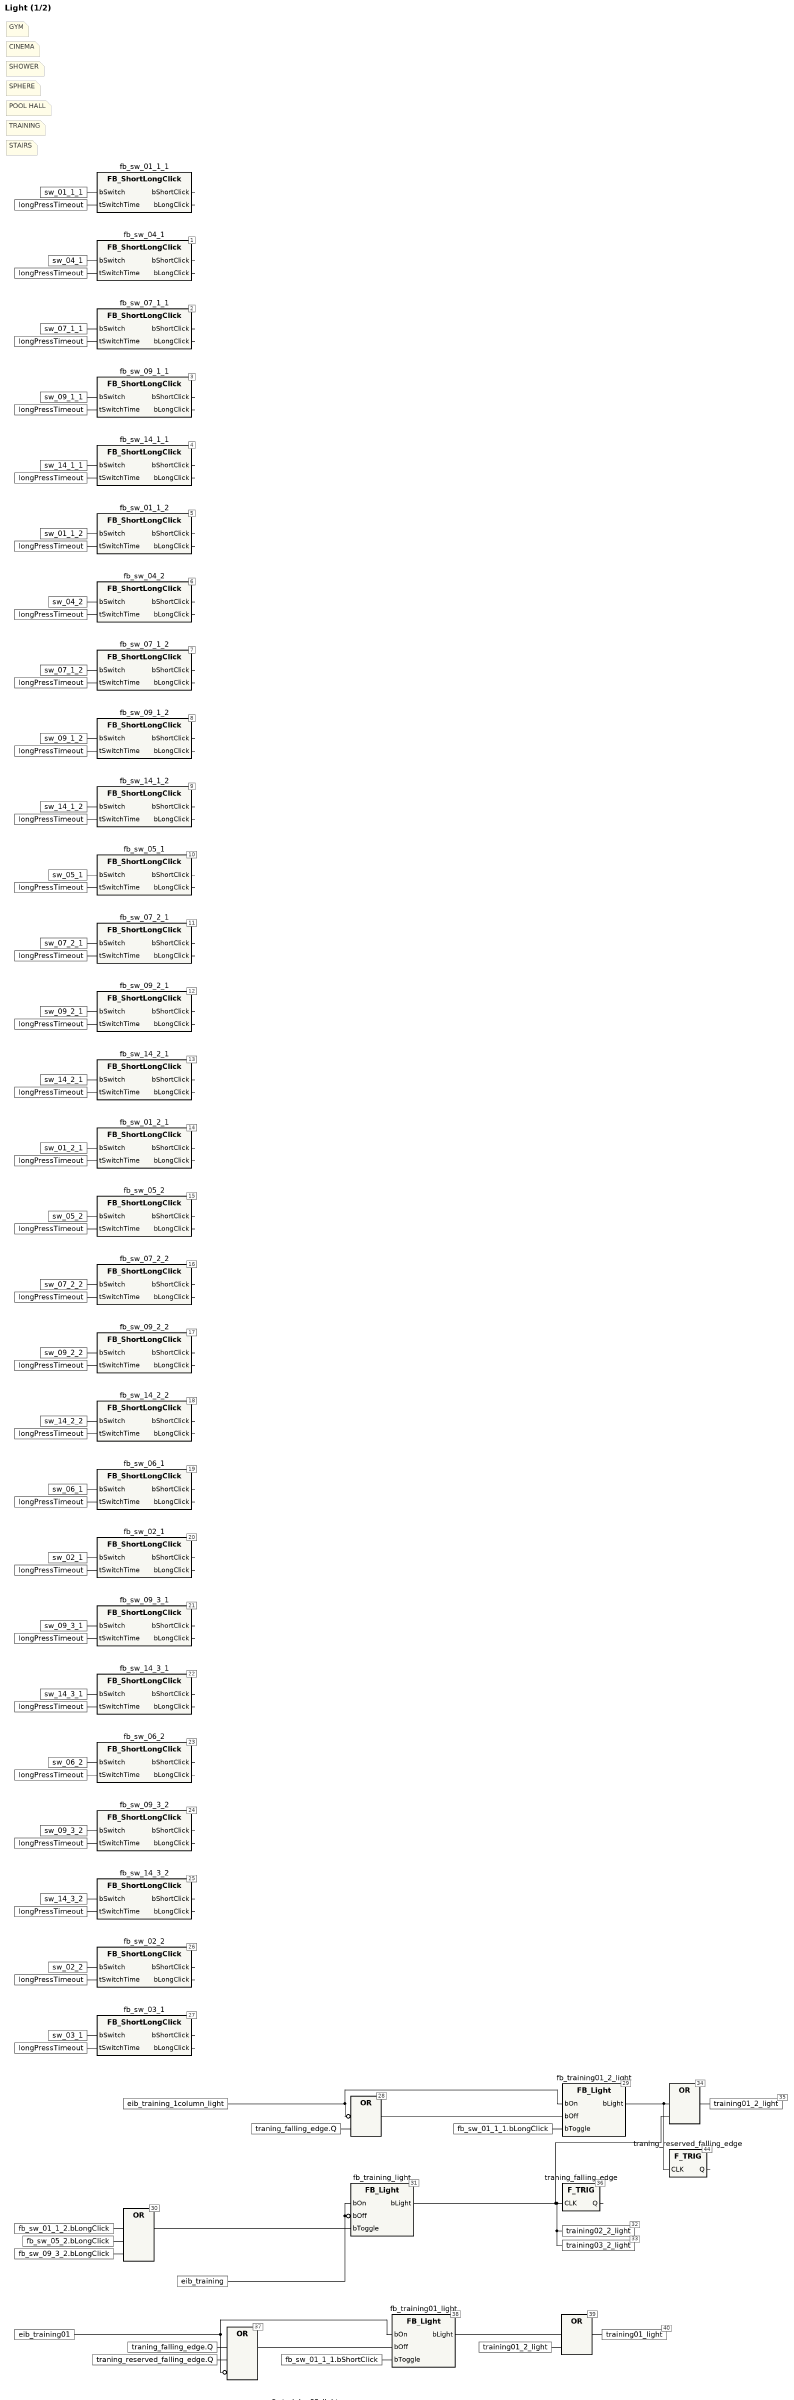
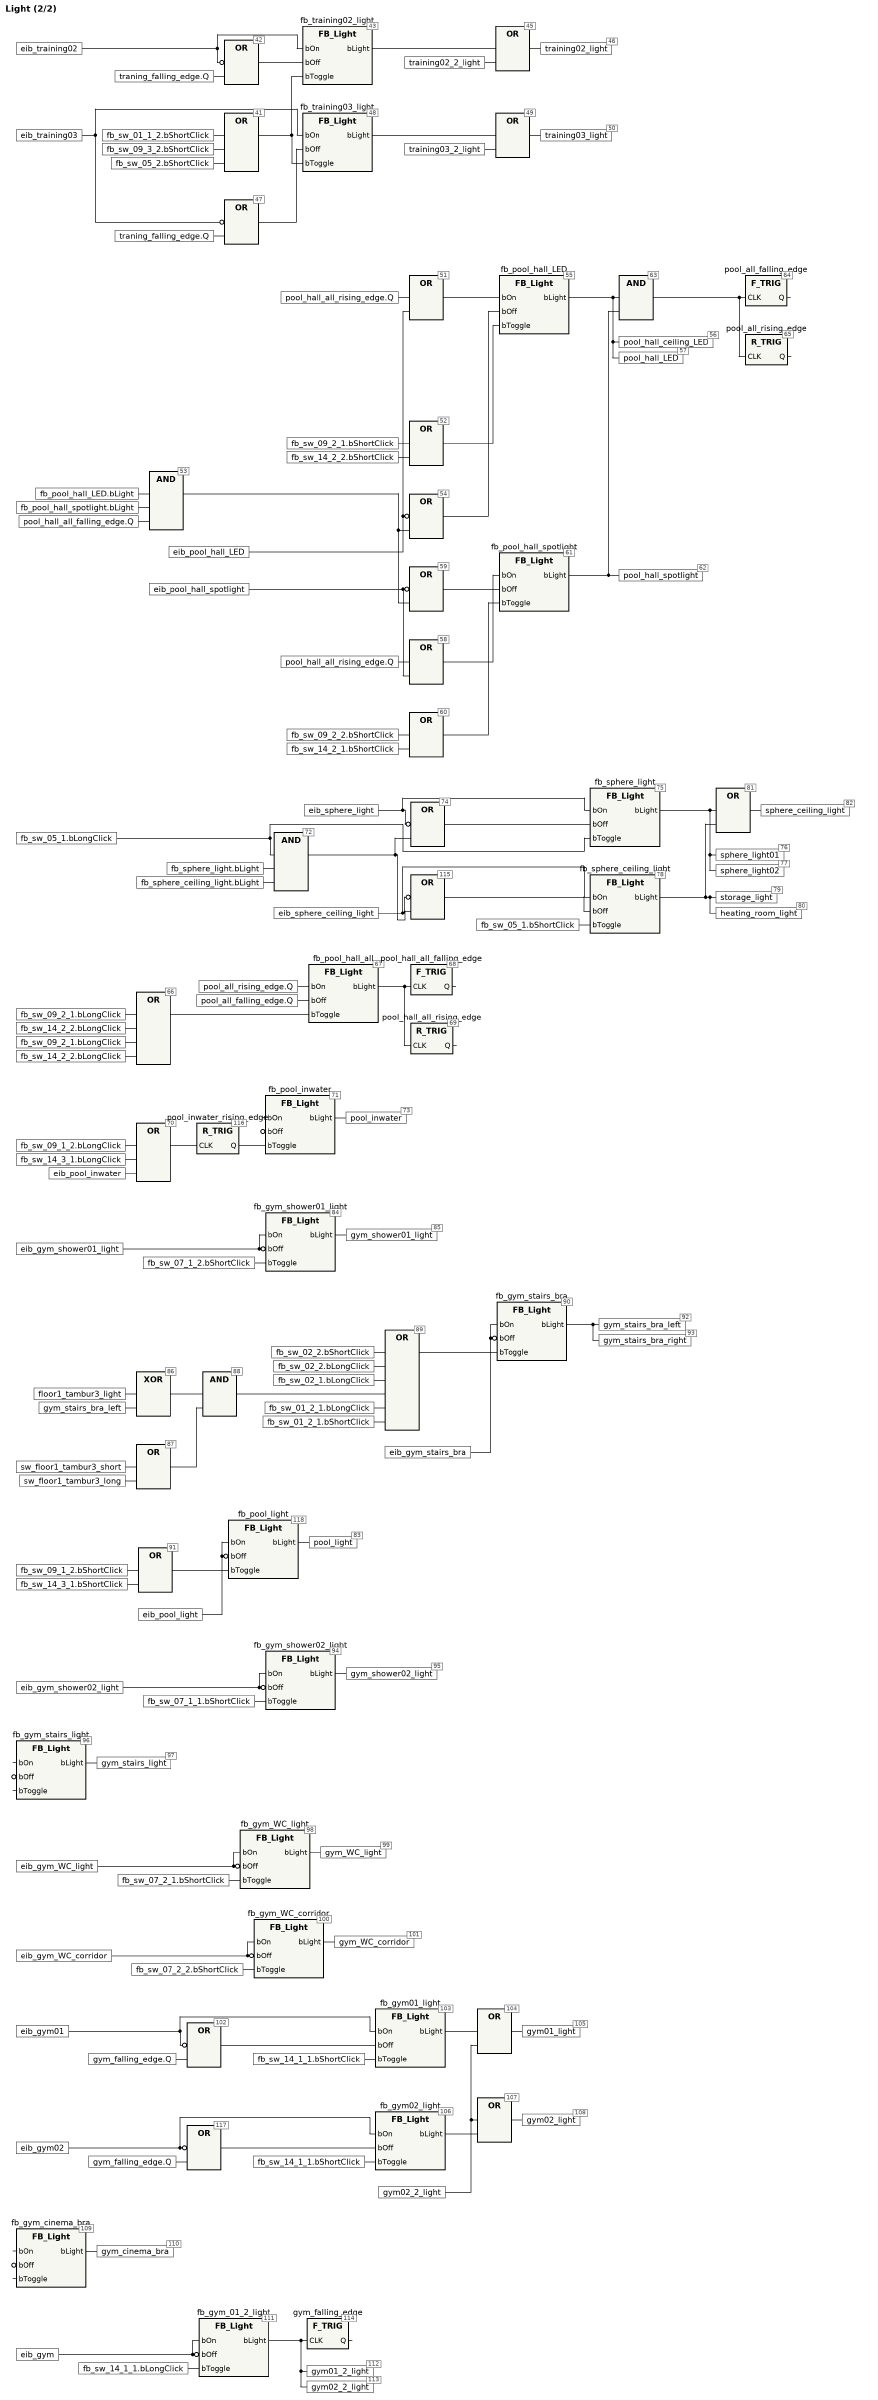
_CFC_ (* Continuous Function Chart, elements in execution order *)
(* GYM *)
(* CINEMA *)
(* SHOWER *)
(* SPHERE *)
(* POOL HALL *)
(* TRAINING *)
(* STAIRS *)
#0 fb_sw_01_1_1:FB_ShortLongClick(bSwitch: sw_01_1_1, tSwitchTime: longPressTimeout)
#1 fb_sw_04_1:FB_ShortLongClick(bSwitch: sw_04_1, tSwitchTime: longPressTimeout)
#2 fb_sw_07_1_1:FB_ShortLongClick(bSwitch: sw_07_1_1, tSwitchTime: longPressTimeout)
#3 fb_sw_09_1_1:FB_ShortLongClick(bSwitch: sw_09_1_1, tSwitchTime: longPressTimeout)
#4 fb_sw_14_1_1:FB_ShortLongClick(bSwitch: sw_14_1_1, tSwitchTime: longPressTimeout)
#5 fb_sw_01_1_2:FB_ShortLongClick(bSwitch: sw_01_1_2, tSwitchTime: longPressTimeout)
#6 fb_sw_04_2:FB_ShortLongClick(bSwitch: sw_04_2, tSwitchTime: longPressTimeout)
#7 fb_sw_07_1_2:FB_ShortLongClick(bSwitch: sw_07_1_2, tSwitchTime: longPressTimeout)
#8 fb_sw_09_1_2:FB_ShortLongClick(bSwitch: sw_09_1_2, tSwitchTime: longPressTimeout)
#9 fb_sw_14_1_2:FB_ShortLongClick(bSwitch: sw_14_1_2, tSwitchTime: longPressTimeout)
#10 fb_sw_05_1:FB_ShortLongClick(bSwitch: sw_05_1, tSwitchTime: longPressTimeout)
#11 fb_sw_07_2_1:FB_ShortLongClick(bSwitch: sw_07_2_1, tSwitchTime: longPressTimeout)
#12 fb_sw_09_2_1:FB_ShortLongClick(bSwitch: sw_09_2_1, tSwitchTime: longPressTimeout)
#13 fb_sw_14_2_1:FB_ShortLongClick(bSwitch: sw_14_2_1, tSwitchTime: longPressTimeout)
#14 fb_sw_01_2_1:FB_ShortLongClick(bSwitch: sw_01_2_1, tSwitchTime: longPressTimeout)
#15 fb_sw_05_2:FB_ShortLongClick(bSwitch: sw_05_2, tSwitchTime: longPressTimeout)
#16 fb_sw_07_2_2:FB_ShortLongClick(bSwitch: sw_07_2_2, tSwitchTime: longPressTimeout)
#17 fb_sw_09_2_2:FB_ShortLongClick(bSwitch: sw_09_2_2, tSwitchTime: longPressTimeout)
#18 fb_sw_14_2_2:FB_ShortLongClick(bSwitch: sw_14_2_2, tSwitchTime: longPressTimeout)
#19 fb_sw_06_1:FB_ShortLongClick(bSwitch: sw_06_1, tSwitchTime: longPressTimeout)
#20 fb_sw_02_1:FB_ShortLongClick(bSwitch: sw_02_1, tSwitchTime: longPressTimeout)
#21 fb_sw_09_3_1:FB_ShortLongClick(bSwitch: sw_09_3_1, tSwitchTime: longPressTimeout)
#22 fb_sw_14_3_1:FB_ShortLongClick(bSwitch: sw_14_3_1, tSwitchTime: longPressTimeout)
#23 fb_sw_06_2:FB_ShortLongClick(bSwitch: sw_06_2, tSwitchTime: longPressTimeout)
#24 fb_sw_09_3_2:FB_ShortLongClick(bSwitch: sw_09_3_2, tSwitchTime: longPressTimeout)
#25 fb_sw_14_3_2:FB_ShortLongClick(bSwitch: sw_14_3_2, tSwitchTime: longPressTimeout)
#26 fb_sw_02_2:FB_ShortLongClick(bSwitch: sw_02_2, tSwitchTime: longPressTimeout)
#27 fb_sw_03_1:FB_ShortLongClick(bSwitch: sw_03_1, tSwitchTime: longPressTimeout)
#28 OR(NOT eib_training_1column_light, traning_falling_edge.Q)
#29 fb_training01_2_light:FB_Light(bOn: eib_training_1column_light, bOff: #28, bToggle: fb_sw_01_1_1.bLongClick)
#30 OR(fb_sw_01_1_2.bLongClick, fb_sw_05_2.bLongClick, fb_sw_09_3_2.bLongClick)
#31 fb_training_light:FB_Light(bOn: eib_training, bOff: NOT eib_training, bToggle: #30)
#32 training02_2_light <= #31.bLight
#33 training03_2_light <= #31.bLight
#34 OR(#29.bLight, #31.bLight)
#35 training01_2_light <= #34
#36 traning_falling_edge:F_TRIG(CLK: #31.bLight)
#37 OR(traning_falling_edge.Q, traning_reserved_falling_edge.Q, NOT eib_training01)
#38 fb_training01_light:FB_Light(bOn: eib_training01, bOff: #37, bToggle: fb_sw_01_1_1.bShortClick)
#39 OR(#38.bLight, training01_2_light)
#40 training01_light <= #39
#41 OR(fb_sw_01_1_2.bShortClick, fb_sw_09_3_2.bShortClick, fb_sw_05_2.bShortClick)
#42 OR(NOT eib_training02, traning_falling_edge.Q)
#43 fb_training02_light:FB_Light(bOn: eib_training02, bOff: #42, bToggle: #41)
#44 traning_reserved_falling_edge:F_TRIG(CLK: #29.bLight)
#45 OR(#43.bLight, training02_2_light)
#46 training02_light <= #45
#47 OR(NOT eib_training03, traning_falling_edge.Q)
#48 fb_training03_light:FB_Light(bOn: eib_training03, bOff: #47, bToggle: #41)
#49 OR(#48.bLight, training03_2_light)
#50 training03_light <= #49
#51 OR(pool_hall_all_rising_edge.Q, eib_pool_hall_LED)
#52 OR(fb_sw_09_2_1.bShortClick, fb_sw_14_2_2.bShortClick)
#53 AND(fb_pool_hall_LED.bLight, fb_pool_hall_spotlight.bLight, pool_hall_all_falling_edge.Q)
#54 OR(NOT eib_pool_hall_LED, #53)
#55 fb_pool_hall_LED:FB_Light(bOn: #51, bOff: #54, bToggle: #52)
#56 pool_hall_ceiling_LED <= #55.bLight
#57 pool_hall_LED <= #55.bLight
#58 OR(pool_hall_all_rising_edge.Q, eib_pool_hall_spotlight)
#59 OR(NOT eib_pool_hall_spotlight, #53)
#60 OR(fb_sw_09_2_2.bShortClick, fb_sw_14_2_1.bShortClick)
#61 fb_pool_hall_spotlight:FB_Light(bOn: #58, bOff: #59, bToggle: #60)
#62 pool_hall_spotlight <= #61.bLight
#63 AND(#55.bLight, #61.bLight)
#64 pool_all_falling_edge:F_TRIG(CLK: #63)
#65 pool_all_rising_edge:R_TRIG(CLK: #63)
#66 OR(fb_sw_09_2_1.bLongClick, fb_sw_14_2_2.bLongClick, fb_sw_09_2_1.bLongClick, fb_sw_14_2_2.bLongClick)
#67 fb_pool_hall_all:FB_Light(bOn: pool_all_rising_edge.Q, bOff: pool_all_falling_edge.Q, bToggle: #66)
#68 pool_hall_all_falling_edge:F_TRIG(CLK: #67.bLight)
#69 pool_hall_all_rising_edge:R_TRIG(CLK: #67.bLight)
#70 OR(fb_sw_09_1_2.bLongClick, fb_sw_14_3_1.bLongClick, eib_pool_inwater)
#71 fb_pool_inwater:FB_Light(bOn: -, bOff: -, bToggle: #116.Q)
#72 AND(fb_sw_05_1.bLongClick, fb_sphere_light.bLight, fb_sphere_ceiling_light.bLight)
#73 pool_inwater <= #71.bLight
#74 OR(NOT eib_sphere_light, #72)
#75 fb_sphere_light:FB_Light(bOn: eib_sphere_light, bOff: #74, bToggle: fb_sw_05_1.bLongClick)
#76 sphere_light01 <= #75.bLight
#77 sphere_light02 <= #75.bLight
#78 fb_sphere_ceiling_light:FB_Light(bOn: eib_sphere_ceiling_light, bOff: #115, bToggle: fb_sw_05_1.bShortClick)
#79 storage_light <= #78.bLight
#80 heating_room_light <= #78.bLight
#81 OR(#75.bLight, #78.bLight)
#82 sphere_ceiling_light <= #81
#83 pool_light <= #118.bLight
#84 fb_gym_shower01_light:FB_Light(bOn: eib_gym_shower01_light, bOff: NOT eib_gym_shower01_light, bToggle: fb_sw_07_1_2.bShortClick)
#85 gym_shower01_light <= #84.bLight
#86 XOR(floor1_tambur3_light, gym_stairs_bra_left)
#87 OR(sw_floor1_tambur3_short, sw_floor1_tambur3_long)
#88 AND(#86, #87)
#89 OR(fb_sw_02_2.bShortClick, fb_sw_02_2.bLongClick, fb_sw_02_1.bLongClick, #88, fb_sw_01_2_1.bLongClick, fb_sw_01_2_1.bShortClick)
#90 fb_gym_stairs_bra:FB_Light(bOn: eib_gym_stairs_bra, bOff: NOT eib_gym_stairs_bra, bToggle: #89)
#91 OR(fb_sw_09_1_2.bShortClick, fb_sw_14_3_1.bShortClick)
#92 gym_stairs_bra_left <= #90.bLight
#93 gym_stairs_bra_right <= #90.bLight
#94 fb_gym_shower02_light:FB_Light(bOn: eib_gym_shower02_light, bOff: NOT eib_gym_shower02_light, bToggle: fb_sw_07_1_1.bShortClick)
#95 gym_shower02_light <= #94.bLight
#96 fb_gym_stairs_light:FB_Light(bOn: -, bOff: -, bToggle: -)
#97 gym_stairs_light <= #96.bLight
#98 fb_gym_WC_light:FB_Light(bOn: eib_gym_WC_light, bOff: NOT eib_gym_WC_light, bToggle: fb_sw_07_2_1.bShortClick)
#99 gym_WC_light <= #98.bLight
#100 fb_gym_WC_corridor:FB_Light(bOn: eib_gym_WC_corridor, bOff: NOT eib_gym_WC_corridor, bToggle: fb_sw_07_2_2.bShortClick)
#101 gym_WC_corridor <= #100.bLight
#102 OR(NOT eib_gym01, gym_falling_edge.Q)
#103 fb_gym01_light:FB_Light(bOn: eib_gym01, bOff: #102, bToggle: fb_sw_14_1_1.bShortClick)
#104 OR(#103.bLight, gym02_2_light)
#105 gym01_light <= #104
#106 fb_gym02_light:FB_Light(bOn: eib_gym02, bOff: #117, bToggle: fb_sw_14_1_1.bShortClick)
#107 OR(gym02_2_light, #106.bLight)
#108 gym02_light <= #107
#109 fb_gym_cinema_bra:FB_Light(bOn: -, bOff: -, bToggle: -)
#110 gym_cinema_bra <= #109.bLight
#111 fb_gym_01_2_light:FB_Light(bOn: eib_gym, bOff: NOT eib_gym, bToggle: fb_sw_14_1_1.bLongClick)
#112 gym01_2_light <= #111.bLight
#113 gym02_2_light <= #111.bLight
#114 gym_falling_edge:F_TRIG(CLK: #111.bLight)
#115 OR(NOT eib_sphere_ceiling_light, #72)
#116 pool_inwater_rising_edge:R_TRIG(CLK: #70)
#117 OR(NOT eib_gym02, gym_falling_edge.Q)
#118 fb_pool_light:FB_Light(bOn: eib_pool_light, bOff: NOT eib_pool_light, bToggle: #91)
_END_CFC_
END_PROGRAM
ACTION knx_triggers:
	rising_edge_eib_gym01 						(CLK:= eib_gym01);
	rising_edge_eib_gym02 						(CLK:= eib_gym02);
	rising_edge_eib_training01 					(CLK:= eib_training01);
	rising_edge_eib_training02						(CLK:=eib_training02 );
	rising_edge_eib_training03						(CLK:= eib_training03);
	rising_edge_eib_gym_stairs_bra				(CLK:= eib_gym_stairs_bra);
	rising_edge_eib_pool_hall_spotlight				(CLK:=eib_pool_hall_spotlight );
	rising_edge_eib_pool_hall_LED				(CLK:= eib_pool_hall_LED);

	rising_edge_eib_pool_light 					(CLK:= eib_pool_light);
	rising_edge_eib_sphere_ceiling_light 			(CLK:= eib_sphere_ceiling_light);
	rising_edge_eib_sphere_light 					(CLK:= eib_sphere_light);
	rising_edge_eib_gym_cinema_bra 				(CLK:= eib_gym_cinema_bra);
	rising_edge_eib_gym_shower01_light			(CLK:= eib_gym_shower01_light);
	rising_edge_eib_gym_shower02_light			(CLK:= eib_gym_shower02_light);
	rising_edge_eib_gym_WC_corridor				(CLK:= eib_gym_WC_corridor);
	rising_edge_eib_gym_stairs_light 				(CLK:= eib_gym_stairs_light);

	rising_edge_eib_gym_WC_light 				(CLK:= eib_gym_WC_light);
	rising_edge_eib_training	 					(CLK:= eib_training);
	rising_edge_eib_gym		 					(CLK:= eib_gym);

	falling_edge_eib_gym01 						(CLK:= eib_gym01);
	falling_edge_eib_gym02 						(CLK:= eib_gym02);
	falling_edge_eib_training01 					(CLK:= eib_training01);
	falling_edge_eib_training02						(CLK:=eib_training02 );
	falling_edge_eib_training03						(CLK:= eib_training03);
	falling_edge_eib_gym_stairs_bra				(CLK:= eib_gym_stairs_bra);
	falling_edge_eib_pool_hall_spotlight				(CLK:=eib_pool_hall_spotlight );
	falling_edge_eib_pool_hall_LED				(CLK:= eib_pool_hall_LED);

	falling_edge_eib_pool_light 					(CLK:= eib_pool_light);
	falling_edge_eib_sphere_ceiling_light 			(CLK:= eib_sphere_ceiling_light);
	falling_edge_eib_sphere_light 					(CLK:= eib_sphere_light);
	falling_edge_eib_gym_cinema_bra 				(CLK:= eib_gym_cinema_bra);
	falling_edge_eib_gym_shower01_light			(CLK:= eib_gym_shower01_light);
	falling_edge_eib_gym_shower02_light			(CLK:= eib_gym_shower02_light);
	falling_edge_eib_gym_WC_corridor				(CLK:= eib_gym_WC_corridor);
	falling_edge_eib_gym_stairs_light 				(CLK:= eib_gym_stairs_light);

	falling_edge_eib_gym_WC_light 				(CLK:= eib_gym_WC_light);
	falling_edge_eib_training	 					(CLK:= eib_training);
	falling_edge_eib_gym		 					(CLK:= eib_gym);
END_ACTION
ACTION outsideLight:
darkOutside_rising_edge(CLK:=bDarkOutside);
IF  darkOutside_rising_edge.Q  THEN
	outside_bigBulbs := TRUE;
	eib_outside_bigBulbs:=TRUE;
	outside_plantsLightning:=TRUE;
	eib_outside_plantsLightning := TRUE;
	outside_smallBulbs := TRUE;
	eib_outside_smallBulbs:= TRUE;
	outside_pingPongTable := FALSE;

ELSE
	outside_bigBulbs := eib_outside_bigBulbs;
	outside_plantsLightning:= eib_outside_plantsLightning;
	outside_smallBulbs := eib_outside_smallBulbs;
	outside_pingPongTable:=eib_outside_pingPongTable;

	IF iHour=0 AND iMinute>=1 AND iMinute<=2 THEN
		outside_bigBulbs := FALSE;
		outside_plantsLightning:=FALSE;
		outside_smallBulbs := FALSE;
		outside_pingPongTable := FALSE;
	END_IF

END_IF;
END_ACTION

(* POU engineering, ST *)
PROGRAM engineering
VAR


END_VAR
pool_floor_heating_pump := eib_pool_floor_heating_pump;
gym_floor_heating_pump := eib_gym_floor_heating_pump;
vent_heating_pump := eib_vent_heating_pump;
heating_pump := eib_heating_pump;
END_PROGRAM

(* POU Counters, ST *)
PROGRAM Counters
VAR

	counter_6_KL1408_1_Input : CTU;

	counter_6_KL1408_3_Input	:	CTU;
	counter_6_KL1408_4_Input	:	CTU;
	counter_6_KL1408_5_Input	:	CTU;
	counter_6_KL1408_6_Input	:	CTU;

	counter_6_KL1408_8_Input	:	CTU;
	counter_7_KL1408_1_Input	:	CTU;
	counter_7_KL1408_2_Input	:	CTU;
	counter_7_KL1408_3_Input	:	CTU;
	counter_7_KL1408_4_Input	:	CTU;
	counter_7_KL1408_5_Input	:	CTU;
	counter_7_KL1408_6_Input	:	CTU;
	counter_7_KL1408_7_Input	:	CTU;
	counter_7_KL1408_8_Input	:	CTU;
	counter_8_KL1408_1_Input	:	CTU;
	counter_8_KL1408_2_Input	:	CTU;
	counter_8_KL1408_3_Input	:	CTU;
	counter_8_KL1408_4_Input	:	CTU;
	counter_8_KL1408_5_Input	:	CTU;
	counter_8_KL1408_6_Input	:	CTU;
	counter_8_KL1408_7_Input	:	CTU;
	counter_8_KL1408_8_Input	:	CTU;
	counter_9_KL1408_1_Input	:	CTU;
	counter_9_KL1408_2_Input	:	CTU;
	counter_9_KL1408_3_Input	:	CTU;
	counter_9_KL1408_4_Input	:	CTU;
	counter_9_KL1408_5_Input	:	CTU;
	counter_9_KL1408_6_Input	:	CTU;
	counter_9_KL1408_7_Input	:	CTU;
	counter_9_KL1408_8_Input	:	CTU;
	counter_10_KL1408_1_Input	:	CTU;
	counter_10_KL1408_2_Input	:	CTU;
	counter_10_KL1408_3_Input	:	CTU;
	counter_10_KL1408_4_Input	:	CTU;
	counter_10_KL1408_5_Input	:	CTU;
	counter_10_KL1408_6_Input	:	CTU;
	counter_10_KL1408_7_Input	:	CTU;
	counter_10_KL1408_8_Input	:	CTU;

	sw01 : INT;
	sw02 : INT;
	sw03 : INT;
	sw04 : INT;
	sw05 : INT;
	sw06 : INT;
	sw07 : INT;
	sw08 : INT;
	sw09 : INT;
	sw10 : INT;
	sw11 : INT;
	sw12 : INT;
	sw13 : INT;
	sw14 : INT;
	sw15 : INT;
	sw16 : INT;
	sw17 : INT;
	sw18 : INT;
	sw19 : INT;
	sw20 : INT;
	sw21 : INT;
	sw22 : INT;
	sw23 : INT;
	sw24 : INT;
	sw25 : INT;
	sw26 : INT;
	sw27 : INT;
	sw28 : INT;
	sw29 : INT;
	sw30 : INT;
	sw31 : INT;
	sw32 : INT;
	sw33 : INT;
	sw34 : INT;
	sw35 : INT;
	sw36 : INT;
	sw37 : INT;
	sw38 : INT;
	sw39 : INT;


END_VAR
	counter_6_KL1408_1_Input(CU:= Term_6_KL1408_1_Input, CV=>sw01);

	counter_6_KL1408_3_Input(CU:= Term_6_KL1408_3_Input, CV=>sw02);
	counter_6_KL1408_4_Input(CU:= Term_6_KL1408_4_Input, CV=>sw03);
	counter_6_KL1408_5_Input(CU:= Term_6_KL1408_5_Input, CV=>sw04);





	counter_7_KL1408_3_Input(CU:= Term_7_KL1408_3_Input, CV=>sw09);

	counter_7_KL1408_5_Input(CU:= Term_7_KL1408_5_Input, CV=>sw11);

	counter_7_KL1408_7_Input(CU:= Term_7_KL1408_7_Input, CV=>sw13);












	counter_9_KL1408_2_Input(CU:= Term_9_KL1408_2_Input, CV=>sw24);

	counter_9_KL1408_4_Input(CU:= Term_9_KL1408_4_Input, CV=>sw26);

	counter_9_KL1408_6_Input(CU:= Term_9_KL1408_6_Input, CV=>sw28);

	counter_9_KL1408_8_Input(CU:= Term_9_KL1408_8_Input, CV=>sw30);

	counter_10_KL1408_1_Input(CU:= Term_10_KL1408_1_Input, CV=>sw31);
	counter_10_KL1408_2_Input(CU:= Term_10_KL1408_2_Input, CV=>sw32);
	counter_10_KL1408_3_Input(CU:= Term_10_KL1408_3_Input, CV=>sw33);
	counter_10_KL1408_4_Input(CU:= Term_10_KL1408_4_Input, CV=>sw34);
	counter_10_KL1408_5_Input(CU:= Term_10_KL1408_5_Input, CV=>sw35);
	counter_10_KL1408_6_Input(CU:= Term_10_KL1408_6_Input, CV=>sw36);
	counter_10_KL1408_7_Input(CU:= Term_10_KL1408_7_Input, CV=>sw37);
	counter_10_KL1408_8_Input(CU:= Term_10_KL1408_8_Input, CV=>sw38);
END_PROGRAM
